FUNCTION_BLOCK Influx2Client (* Template for a Simple Function Block Type *)
  (* Standard: 61499-1 *)
  (* Version 1.0, 2024-08-01, david *)
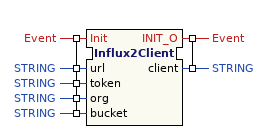
  EVENT_INPUT
    Init WITH url, token, org, bucket; (* Initialze Function Block *)
  END_EVENT
  EVENT_OUTPUT
    INIT_O WITH client; (* Execution Confirmation *)
  END_EVENT
  VAR_INPUT
    url : STRING; (* Input *)
    token : STRING; (* Access token of Database *)
    org : STRING; (* Organisation *)
    bucket : STRING; (* Data bucket *)
  END_VAR
  VAR_OUTPUT
    client : STRING; (* Client object *)
  END_VAR
  ALGORITHM REQ IN ST: (* Normally executed algorithm *)
OUT := IN;
  END_ALGORITHM
END_FUNCTION_BLOCK
